INTERFACE I_Disposable EXTENDS I_Base

METHOD Dispose
VAR_INPUT
END_VAR
END_METHOD

END_INTERFACE

(* stored: Version 1.1.0.1, ProductVersion 3.1.4026.18
   Itf I_Disposable: Id {7257362c-a4db-4e4f-ad30-a830a19d60e9}
   Method Dispose: Id {2ac932df-7230-4007-b636-6f144e772cee} *)
